// /////////////////////////////////////////////////////////////////////////////
// ///                                                                       ///
// ///    SYSTEM:     AIRPORT EMERGENCY DOOR                                 ///
// ///                                                                       ///
// ///                                                                       ///
// ///    SUBJECT:       AUTOMATION AND INDUSTRIAL INSTRUMENTATION           ///
// ///    DATE:       2026-04-01                                             ///
// ///                                                                       ///
// ///    MADE BY:    [01] Iñigo Bañuls                                      ///
// ///                [02] Lander Nieto                                      ///
// ///                [03] Ruud Rohan                                        ///
// ///                                                                       ///
// /////////////////////////////////////////////////////////////////////////////



PROGRAM MAIN
VAR
	{attribute 'OPC.UA.DA' := '1'}
	stSystem	:	sysType;                  // SYSTEM DATA STRUCT
	EMERGENCY_HDL	: FB_EMERGENCY_SYS;		  // EMERGENCY HANDLING FUNCTION BLOCK	
	RPi_WATCHDOG	: FB_RPi_WATCHDOG;
	
	STEPPER_CTRL    : FB_STEPPER_CTRL;		  // STEPPER MOTOR CONTROL
    bIsOpening      : BOOL;
    bIsClosing      : BOOL;
	
// Atributos para exponer las variables al servidor OPC UA
    {attribute 'OPC.UA.DA' := '1'}
    aImageRxBuffer : ARRAY[0..99999] OF BYTE; // Buffer para recibir desde la RPi (Ej: 100 KB)
    
    {attribute 'OPC.UA.DA' := '1'}
    aImageTxBuffer : ARRAY[0..99999] OF BYTE; // Buffer para enviar a la RPi
    
    // Variables de control (Handshake)
    {attribute 'OPC.UA.DA' := '1'}
    bRpiHasWritten : BOOL; // La RPi lo pone en TRUE cuando termina de enviar
    
    {attribute 'OPC.UA.DA' := '1'}
    bPlcHasWritten : BOOL; // El PLC lo pone en TRUE cuando tiene una imagen lista para la RPi

END_VAR

EMERGENCY_HDL(stSystem := stSystem);
RPi_WATCHDOG(stSystem := stSystem);
EMERGENCY_HDL.mTransitions(stSystem := stSystem);

// 1. Evaluamos si la máquina de estados está en un estado de APERTURA
bIsOpening := (stSystem.state = sysState.stOpening) OR
              (stSystem.state = sysState.stAlarmOpening) OR
              (stSystem.state = sysState.stFaceDetectionAlarmOpening) OR
              (stSystem.state = sysState.stConfigOpening) OR
              (stSystem.state = sysState.stRaspberryFailOpening);

// 2. Evaluamos si la máquina de estados está en un estado de CIERRE
bIsClosing := (stSystem.state = sysState.stClosing) OR
              (stSystem.state = sysState.stAlarmClosing) OR
              (stSystem.state = sysState.stFaceDetectionAlarmClosing) OR
              (stSystem.state = sysState.stConfigClosing);

// 3. Llamada al controlador del motor paso a paso
// El motor girará continuamente mientras bIsOpening o bIsClosing sean TRUE.
// Se detendrá (reseteando pulsos) cuando la máquina pase a un estado estático (ej. stAlarm, stRaspberryOk, etc.)
STEPPER_CTRL(
    bOpen   := bIsOpening,
    bClose  := bIsClosing,
    bEnable := TRUE, // Puedes condicionar esto a (stSystem.state <> sysState.stDisconnected) si lo prefieres
    bPulse  => stSystem.outputs.oMotorPulse,
    bDir    => stSystem.outputs.oMotorDir
);

END_PROGRAM

(* stored: Version 1.1.0.1, ProductVersion 3.1.4026.12
   POU MAIN: Id {1185f6f7-1cbe-454c-8e29-f938133bda08}, SpecialFunc None *)
